FUNCTION_BLOCK XTSIOEnvVarWrapper IMPLEMENTS ITF_XTSIOEnvVarWrapper
VAR
	XtsIoEnvironment : Tc3_XTS_Utility.FB_TcIoXtsEnvironment;
	stXtsEnvironmentConfiguration	: ST_XtsEnvironmentConfiguration;
	XPU: Tc3_XTS_Utility.I_TcIoXtsProcessingUnit;
	Initialised : BOOL;
END_VAR

METHOD FB_init : BOOL
VAR_INPUT
	bInitRetains : BOOL; // if TRUE, the retain variables are initialized (warm start / cold start)
	bInCopyCode : BOOL;  // if TRUE, the instance afterwards gets moved into the copy code (online change)
END_VAR
stXtsEnvironmentConfiguration.bEnableInitCaGroup := TRUE;
XtsIoEnvironment.P_XtsEnvironmentConfiguration := stXtsEnvironmentConfiguration;
END_METHOD

METHOD GetCaGroupInterface : I_Mc2CaGroup
VAR_INPUT
	CAGroupNumber : INT;
END_VAR
GetCaGroupInterface := XtsIoEnvironment.Mc2CaGroup(1);
END_METHOD

METHOD PUBLIC GetMotorModuleInterface : I_TcIoXtsPartModule
VAR_INPUT
	PartNumber : INT;
	ModuleNumber : INT;
END_VAR
XPU.PartTcIo(PartNumber).ModuleTcIo(ModuleNumber);
END_METHOD

METHOD PUBLIC GetMoverInterface : I_TcIoXtsXpuMover
VAR_INPUT
	MoverId : INT;
END_VAR
GetMoverInterface := XPU.MoverTcIo(MoverID);
END_METHOD

METHOD PUBLIC GetPartInterface : I_TcIoXtsXpuPart
VAR_INPUT
	PartNumber : INT;
END_VAR
GetPartInterface := XPU.PartTcIo(PartNumber);
END_METHOD

METHOD PUBLIC GetTrackInterface : I_TcIoXtsXpuTrack
VAR_INPUT
	TrackNumber : INT;
END_VAR
GetTrackInterface := XPU.TrackTcIo(TrackNumber);
END_METHOD

METHOD GetXPUInterface : I_TcIoXtsProcessingUnit
VAR_INPUT
END_VAR
GetXPUInterface := XPU;
END_METHOD

METHOD PUBLIC Initialise : BOOL
VAR_INPUT
END_VAR
IF XtsIoEnvironment.Init(TRUE) THEN
	XtsIoEnvironment.Init(FALSE);
	XPU := XtsIoEnvironment.XpuTcIo(1);
	Initialise := Initialised := TRUE;
END_IF
END_METHOD

METHOD IsInitialised : BOOL
VAR_INPUT
END_VAR
IsInitialised := Initialised;
END_METHOD

METHOD IsInSim : BOOL
VAR_INPUT
END_VAR
IF  XPU.GetOperationMode() = OperationMode.Simulation THEN
	IsInSim := TRUE;
END_IF
END_METHOD

METHOD TriggerDetection : BOOL
VAR_INPUT
END_VAR
XPU.TriggerDetection();
TriggerDetection := true;
END_METHOD

METHOD TriggerRedetection : BOOL
VAR_INPUT
END_VAR
TriggerRedetection := XPU.TriggerRedetection();
END_METHOD

END_FUNCTION_BLOCK

(* stored: Version 1.1.0.1, ProductVersion 3.1.4026.11
   POU XTSIOEnvVarWrapper: Id {03c3c931-6ee3-4ab9-88b9-320f3e1d8e15}, SpecialFunc None
   Method FB_init: Id {5798f5d6-785a-4124-98b0-b4ab031dfdac}
   Method GetCaGroupInterface: Id {12f834a0-9ae6-48b5-9bae-7bc717cd2b2d}
   Method GetMotorModuleInterface: Id {9af7c768-b524-4dfc-b4c9-d134e43969ae}
   Method GetMoverInterface: Id {dbc9b774-d169-476b-835b-9bf55e4a60d9}
   Method GetPartInterface: Id {a60c8186-f31f-4591-b959-ebb1bad32c7a}
   Method GetTrackInterface: Id {36334a76-598d-4a99-aaef-0a407eed48bd}
   Method GetXPUInterface: Id {a6b4198a-d372-4fc0-b700-debb44563dc0}
   Method Initialise: Id {f0d17991-21f7-403c-899a-0fcccbff041e}
   Method IsInitialised: Id {66e54d32-1c95-4eb4-ba62-654c54ac7108}
   Method IsInSim: Id {4972b79f-8f9e-49c6-8407-5f314a09a94a}
   Method TriggerDetection: Id {1bac5fa5-b8a9-4a64-8a15-4af89462d3b7}
   Method TriggerRedetection: Id {ae4a38c2-59c8-4f6f-9609-030adeda16ad} *)
